{library PUBLIC}
(*
Get progress value for ASync calls.
This function block will read the global status.
To see a specific function progress use the output of RPCx or ASyncRP function blocks.
*)

FUNCTION_BLOCK ASyncProgress
VAR_INPUT
	En: 				BOOL;			(* Set to true to get progress value *)
END_VAR
VAR_OUTPUT
	Done:				BOOL;			(* Done = En *)
	Progress: 			INT;			(* Progress value *)
END_VAR
VAR_IN_OUT
	Data: 				CommunicationData;		(* Common data structure to connect this function block to a specific Communicator block *)
END_VAR
VAR
END_VAR

IF En THEN
	Progress:=Data._ASyncProgress;
ELSE
	Progress:=0;
END_IF;

Done:=En;

END_FUNCTION_BLOCK

(* stored: Version 1.1.0.1, ProductVersion 3.1.4024.2
   POU ASyncProgress: Id {65dd0780-74ba-4325-af35-64ebb6ab86de}, SpecialFunc None *)
